PROGRAM PrgMqttCom
VAR
	fbMqttClient : FB_IotMqttClient;
	bSetParameter : BOOL := TRUE;
	bConnect : BOOL := TRUE;
	
	sTopicPub : STRING(255) := 'MyTopic';
	sPayloadPub : STRING(255) := 'Hello from TwinCAT';
	i: UDINT;
	fbTimer : TON := (PT:=T#1S);
	
	hrErrorOccurred : HRESULT; // contains the latest occurred error
END_VAR
VAR CONSTANT	
	cMyPskKey : ARRAY[1..64] OF BYTE := [16#1B, 16#D0, 16#6F, 16#D2, 16#56, 16#16, 16#7D, 16#C1, 16#E8, 16#C7, 16#48, 16#2A, 16#8E, 16#F5, 16#FF];
END_VAR

IF bSetParameter THEN
	bSetParameter := FALSE;

	fbMqttClient.stTLS.sPskIdentity := 'my_Identity';
	fbMqttClient.stTLS.aPskKey := cMyPskKey;
	fbMqttClient.stTLS.nPskKeyLen := 15;		
	fbMqttClient.nHostPort := 8883;
END_IF

fbMqttClient.Execute(bConnect);
IF fbMqttClient.bError THEN
	// add your error logging here
	hrErrorOccurred := fbMqttClient.hrErrorCode;
END_IF

IF fbMqttClient.bConnected THEN
	fbTimer(IN:=TRUE);
	IF fbTimer.Q THEN // publish new payload every second
		fbTimer(IN:=FALSE);
		i := i + 1;
		sPayloadPub := CONCAT('MyMessage', TO_STRING(i));
		fbMqttClient.Publish(	sTopic:= sTopicPub, 
								pPayload:= ADR(sPayloadPub), nPayloadSize:= LEN2(ADR(sPayloadPub))+1, 
								eQoS:= TcIotMqttQos.AtMostOnceDelivery, bRetain:= FALSE, bQueue:= FALSE );
		IF fbMqttClient.bError THEN
			// add your error logging here
			hrErrorOccurred := fbMqttClient.hrErrorCode;
		END_IF
	END_IF
END_IF

END_PROGRAM

(* stored: Version 1.1.0.1, ProductVersion 3.1.4022.3
   POU PrgMqttCom: Id {c70f107a-6ca5-4bfb-b775-e2929cbf9dae}, SpecialFunc None *)
